ABB RobotStudio station: conveier tracking_assingment(incomplet(error)).rsstn

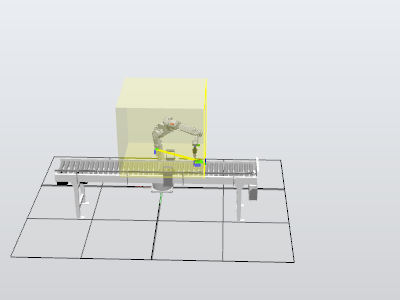
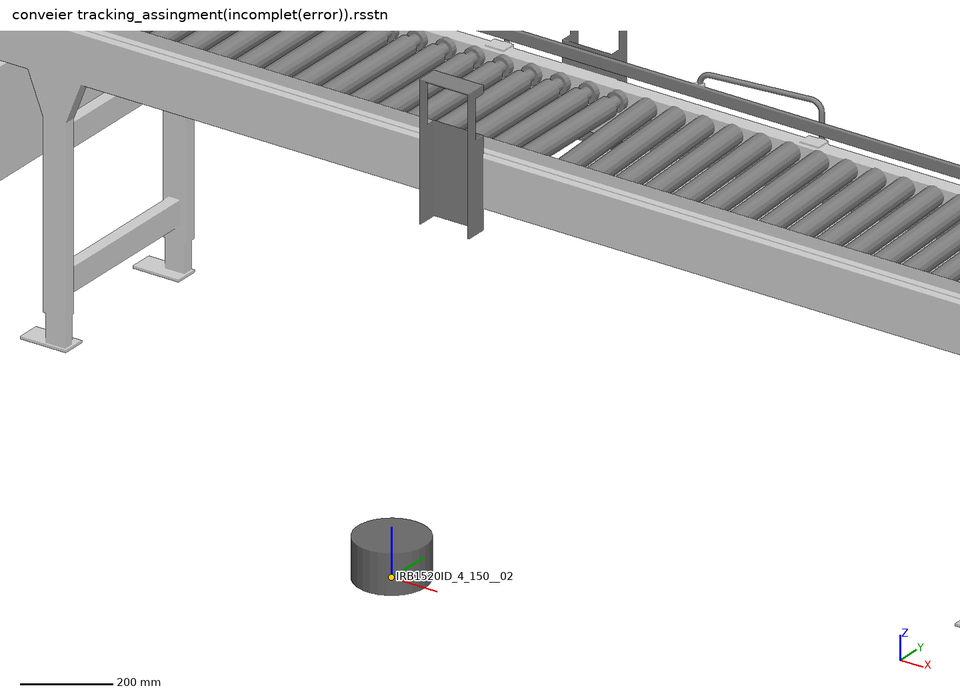
[picture v1: parts stored in the station drawn from their meshes, with robot base, taught points and paths (robot models come from the ABB library and are not in the file)]
Station Station (saved by RobotStudio 22.3.10141.1)
Controller Controller29, task T_ROB1: task frame (RAPID world) sits at (-710.04, 543.58, 775) mm in the station
Controller Controller29
  mechanical unit ROB_1: IRB1520ID_4_150__02, 6 joints, base frame (710.04, -543.58, -775) mm, rotated rx 0 ry 0 rz 90 deg
  mechanical unit CNV1: ?, 1 joints, base frame (0, 0, 0) mm
Layout (positions relative to the parent item):
  - IRB1520ID_4_150__02 [mechanism, from Robots\IRB1520ID_4_150_G_02.rslib] at (0, 0, 0) mm, rotated rx 0 ry 0 rz 90 deg; joint values [0.8536, -0.221, 0.1715, -0.5187, 1.1979, 0.9413] (rad or m)
  - MyTool [mechanism, from Training Objects\myTool.rslib] at (-560.05, 610.96, 1106.28) mm, rotated rx 179.91 ry 37.84 rz -90.06 deg
  - Conveyor [conveyor]
    - 400_guide [part] at (-1484.89, 541.08, 0) mm, size 3033 x 590 x 945 mm
    - Part_1 [part], size 176 x 175.7 x 100 mm
Attachment: MyTool is attached to IRB1520ID_4_150__02 / Link6
Conveyor tracking Connection: unit CNV1, TravelOffset=0.7, QueueTrackDistance=0, StartWindowWidth=1.25, SyncSeparation=0.1, CountsPerMeter=10000
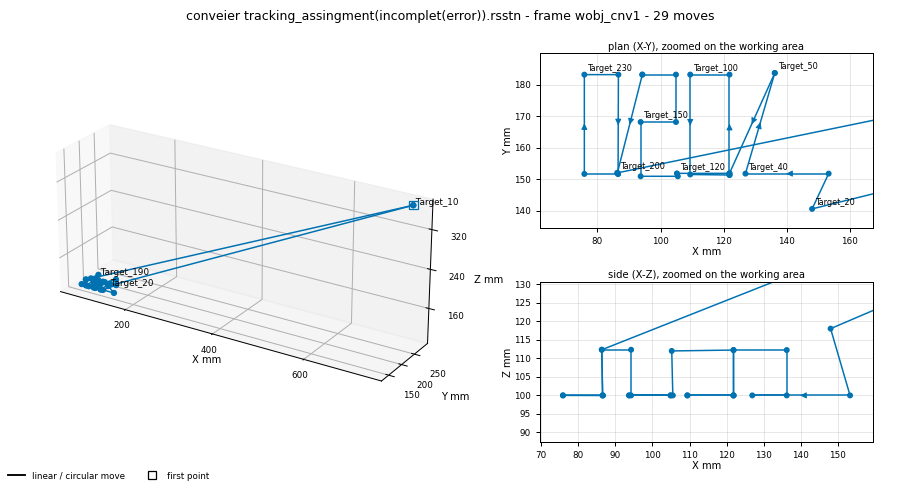
[picture p0: tool path of conveier tracking_assingment(incomplet(error)).rsstn in frame wobj_cnv1, 29 of 29 moves have a stored position in this frame; points joined in program order, loops and branches not executed]
Targets, tools, work objects and paths stored in the station, written as RAPID:
! task T_ROB1
MODULE CalibData
  PERS tooldata MyTool:=[TRUE,[[31.792631019,0,229.638935148],[0.945518576,0,0.325568154,0]],[1,[0,0,1],[1,0,0,0],0,0,0]];
  TASK PERS wobjdata wobj_cnv1:=[FALSE,FALSE,"CNV1",[[0,0,0],[1,0,0,0]],[[0,0,0],[1,0,0,0]]];
ENDMODULE

! task T_ROB1
MODULE Module1
  CONST robtarget Target_10:=[[732.463009475,284.74015252,367.850986194],[0.134921751,-0.694115329,0.694115379,0.134921726],[-1,0,-1,0],[9E+09,9E+09,9E+09,9E+09,9E+09,0]];
  CONST robtarget Target_20:=[[148.027259086,140.620270023,118.002263215],[0.001426554,0.707106573,-0.70710535,0.000532065],[0,-1,0,0],[9E+09,9E+09,9E+09,9E+09,9E+09,0]];
  CONST robtarget Target_30:=[[153.26852847,151.790865361,99.999975909],[0.001426762,0.707106584,-0.707105338,0.000532256],[0,-1,0,0],[9E+09,9E+09,9E+09,9E+09,9E+09,0]];
  CONST robtarget Target_40:=[[126.907111414,151.790839328,99.999990319],[0.001426849,0.707106584,-0.707105338,0.000532331],[0,-1,0,0],[9E+09,9E+09,9E+09,9E+09,9E+09,0]];
  CONST robtarget Target_50:=[[136.201780371,183.668259016,99.999982831],[0.001427063,0.707106549,-0.707105373,0.000532586],[0,-1,0,0],[9E+09,9E+09,9E+09,9E+09,9E+09,0]];
  CONST robtarget Target_60:=[[136.201785973,183.668257816,112.228065217],[0.001427184,0.707106531,-0.70710539,0.000532738],[0,-1,0,0],[9E+09,9E+09,9E+09,9E+09,9E+09,0]];
  CONST robtarget Target_70:=[[121.84807836,151.875094498,112.228069099],[0.001427329,0.707106549,-0.707105372,0.000532907],[0,-1,0,0],[9E+09,9E+09,9E+09,9E+09,9E+09,0]];
  CONST robtarget Target_80:=[[121.85294123,151.351761703,99.999985623],[0.001427546,0.707106545,-0.707105376,0.000533146],[0,-1,0,0],[9E+09,9E+09,9E+09,9E+09,9E+09,0]];
  CONST robtarget Target_90:=[[121.852970197,183.165253797,99.999984063],[0.001427623,0.70710654,-0.70710538,0.000533249],[0,-1,0,0],[9E+09,9E+09,9E+09,9E+09,9E+09,0]];
  CONST robtarget Target_100:=[[109.410061468,183.165252044,99.999998854],[0.001427674,0.707106564,-0.707105356,0.000533323],[0,-1,0,0],[9E+09,9E+09,9E+09,9E+09,9E+09,0]];
  CONST robtarget Target_110:=[[109.410077867,151.516573695,99.999994682],[0.001427712,0.707106561,-0.707105359,0.000533354],[0,-1,0,0],[9E+09,9E+09,9E+09,9E+09,9E+09,0]];
  CONST robtarget Target_120:=[[105.194212502,151.875183004,111.988869677],[0.001427517,0.70710657,-0.707105351,0.000533104],[0,-1,0,0],[9E+09,9E+09,9E+09,9E+09,9E+09,0]];
  CONST robtarget Target_130:=[[105.485840783,150.946217613,99.999987102],[0.001427757,0.707106621,-0.707105299,0.000533301],[0,-1,0,0],[9E+09,9E+09,9E+09,9E+09,9E+09,0]];
  CONST robtarget Target_140:=[[93.698227672,150.946256037,99.999984545],[0.001427954,0.707106618,-0.707105301,0.000533487],[0,-1,0,0],[9E+09,9E+09,9E+09,9E+09,9E+09,0]];
  CONST robtarget Target_150:=[[93.698238522,168.144158754,99.999989888],[0.001427971,0.707106631,-0.707105289,0.000533554],[0,-1,0,0],[9E+09,9E+09,9E+09,9E+09,9E+09,0]];
  CONST robtarget Target_160:=[[104.886729994,168.144147259,99.999983588],[0.00142803,0.707106618,-0.707105301,0.000533604],[0,-1,0,0],[9E+09,9E+09,9E+09,9E+09,9E+09,0]];
  CONST robtarget Target_170:=[[104.886725613,183.161493982,99.9999804],[0.001428121,0.707106621,-0.707105298,0.0005337],[0,-1,0,0],[9E+09,9E+09,9E+09,9E+09,9E+09,0]];
  CONST robtarget Target_180:=[[94.233944248,183.161507641,99.999991636],[0.001428155,0.707106639,-0.70710528,0.000533738],[0,-1,0,0],[9E+09,9E+09,9E+09,9E+09,9E+09,0]];
  CONST robtarget Target_190:=[[94.233923745,183.16155166,112.314908633],[0.001428246,0.707106642,-0.707105277,0.000533805],[0,-1,0,0],[9E+09,9E+09,9E+09,9E+09,9E+09,0]];
  CONST robtarget Target_200:=[[86.332966166,152.035065737,112.314897532],[0.001428381,0.707106621,-0.707105297,0.000533909],[0,-1,0,0],[9E+09,9E+09,9E+09,9E+09,9E+09,0]];
  CONST robtarget Target_210:=[[86.550308991,151.694086969,99.999995992],[0.001428538,0.70710656,-0.707105358,0.000534084],[0,-1,0,0],[9E+09,9E+09,9E+09,9E+09,9E+09,0]];
  CONST robtarget Target_220:=[[75.865021826,151.694059196,99.999983948],[0.001428621,0.707106566,-0.707105352,0.000534181],[0,-1,0,0],[9E+09,9E+09,9E+09,9E+09,9E+09,0]];
  CONST robtarget Target_230:=[[75.864806695,183.153257867,99.999985123],[0.001428716,0.707106581,-0.707105336,0.00053427],[0,-1,0,0],[9E+09,9E+09,9E+09,9E+09,9E+09,0]];
  CONST robtarget Target_240:=[[86.654880498,183.153292005,99.974308059],[0.001428804,0.707106564,-0.707105353,0.000534358],[0,-1,0,0],[9E+09,9E+09,9E+09,9E+09,9E+09,0]];
  PROC Path_10()
    ActUnit CNV1;
    WaitWObj wobj0\MaxTime:=0.5;
    MoveL Target_10,v1000,z100,MyTool\WObj:=wobj_cnv1;
    MoveL Target_20,v1000,z100,MyTool\WObj:=wobj_cnv1;
    MoveL Target_30,v1000,z100,MyTool\WObj:=wobj_cnv1;
    MoveL Target_40,v1000,z100,MyTool\WObj:=wobj_cnv1;
    MoveL Target_50,v1000,z100,MyTool\WObj:=wobj_cnv1;
    MoveL Target_60,v1000,z100,MyTool\WObj:=wobj_cnv1;
    MoveL Target_70,v1000,z100,MyTool\WObj:=wobj_cnv1;
    MoveL Target_80,v1000,z100,MyTool\WObj:=wobj_cnv1;
    MoveL Target_90,v1000,z100,MyTool\WObj:=wobj_cnv1;
    MoveL Target_100,v1000,z100,MyTool\WObj:=wobj_cnv1;
    MoveL Target_110,v1000,z100,MyTool\WObj:=wobj_cnv1;
    MoveL Target_80,v1000,z100,MyTool\WObj:=wobj_cnv1;
    MoveL Target_70,v1000,z100,MyTool\WObj:=wobj_cnv1;
    MoveL Target_120,v1000,z100,MyTool\WObj:=wobj_cnv1;
    MoveL Target_130,v1000,z100,MyTool\WObj:=wobj_cnv1;
    MoveL Target_140,v1000,z100,MyTool\WObj:=wobj_cnv1;
    MoveL Target_150,v1000,z100,MyTool\WObj:=wobj_cnv1;
    MoveL Target_160,v1000,z100,MyTool\WObj:=wobj_cnv1;
    MoveL Target_170,v1000,z100,MyTool\WObj:=wobj_cnv1;
    MoveL Target_180,v1000,z100,MyTool\WObj:=wobj_cnv1;
    MoveL Target_190,v1000,z100,MyTool\WObj:=wobj_cnv1;
    MoveL Target_200,v1000,z100,MyTool\WObj:=wobj_cnv1;
    MoveL Target_210,v1000,z100,MyTool\WObj:=wobj_cnv1;
    MoveL Target_220,v1000,z100,MyTool\WObj:=wobj_cnv1;
    MoveL Target_230,v1000,z100,MyTool\WObj:=wobj_cnv1;
    MoveL Target_240,v1000,z100,MyTool\WObj:=wobj_cnv1;
    MoveL Target_210,v1000,z100,MyTool\WObj:=wobj_cnv1;
    MoveL Target_200,v1000,z100,MyTool\WObj:=wobj_cnv1;
    MoveL Target_10,v1000,z100,MyTool\WObj:=wobj_cnv1;
    WaitWObj wobj0\MaxTime:=0.5;
  ENDPROC
ENDMODULE

